(* LS Electric XG5000 project: 06_Practice_Questions *)
(* PLC LSPLC *)
(* module base 0 slot 0: 입력 모듈:XGI-D21A (DC 24V 입력, 8점 (전류소스/싱크입력)) *)
(* module base 0 slot 1: 출력 모듈:XGQ-RY1A (릴레이 출력, 8점 (2A용, 단독 COM.)) *)

PROGRAM NewProgram (* task: 스캔 프로그램 *)
VAR
    Flipflop : FF;
    Flipflop1 : FF;
    P0 AT %IX0.0.0 : BOOL;
    P1 AT %IX0.0.1 : BOOL;
    P10 AT %QX0.1.0 : BOOL;
    P11 AT %QX0.1.1 : BOOL;
    P12 AT %QX0.1.2 : BOOL;
    P2 AT %IX0.0.2 : BOOL;
    P3 AT %IX0.0.3 : BOOL;
    곱셈결과 : INT;
    곱셈결과2 : UDINT;
    메모리0 AT %MX0 : BOOL;
    시간 : TIME;
    시간_중간 : UDINT;
    시작 : BOOL;
    업카운터 : CTD_INT;
    천 : INT := 1000;
    카운터 : CTU_INT;
    카운터1 : CTU_INT;
    카운트 : INT;
    타이머1 : TP;
    타이머2 : TP;
    타이머3 : TP;
END_VAR

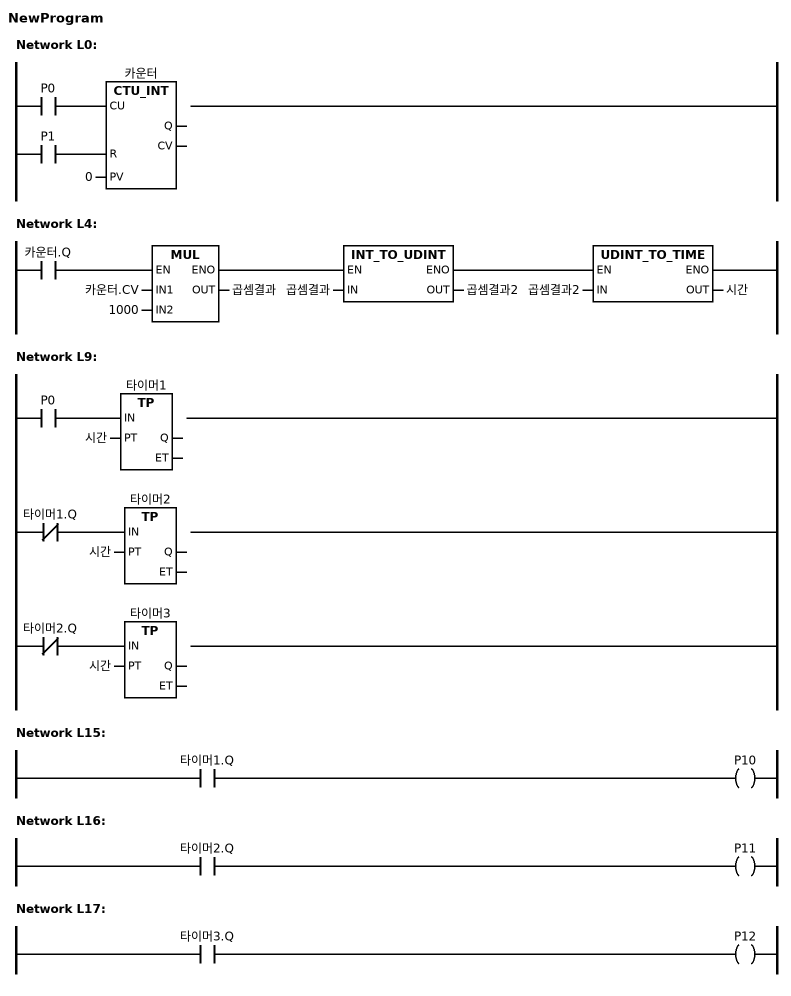
(* Rung L0 *)
카운터(CU := P0, R := P1, PV := 0);
(* Rung L4 *)
IF 카운터.Q THEN
    곱셈결과 := 카운터.CV * 1000;
    곱셈결과2 := INT_TO_UDINT(곱셈결과);
    시간 := UDINT_TO_TIME(곱셈결과2);
END_IF;
(* Rung L9 *)
타이머1(IN := P0, PT := 시간);
타이머2(IN := NOT 타이머1.Q, PT := 시간);
타이머3(IN := NOT 타이머2.Q, PT := 시간);
(* Rung L15 *)
P10 := 타이머1.Q;
(* Rung L16 *)
P11 := 타이머2.Q;
(* Rung L17 *)
P12 := 타이머3.Q;
END_PROGRAM